Staubli VAL3: park1.pgx

program park1()
begin
  // -- move back to rest position
  resetMotion()
  movej(jRestPosition,tTool,mNomSpeed)
  waitEndMove()
end
